FUNCTION_BLOCK AQ_SPLIT_2 (* Fan-Out: Splits 1 AQ into 2 AQ adapters *)
  (* Standard: 61499-2; Description: Copyright (c) 2026 Meisterschulen am Ostbahnhof SPDX-License-Identifier: EPL-2.0 *)
  (* Version 1.0, 2026-05-16, Franz Höpfinger, Meisterschulen am Ostbahnhof, Initial Version *)
  PACKAGE adapter::events::unidirectional;
  IMPORT eclipse4diac::core::GenericClassName;
  {SET_ATTRIBUTE(eclipse4diac::core::GenericClassName, 'GEN_AQ_SPLIT')}
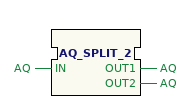
  SOCKETS
    IN : adapter::types::unidirectional::AQ; (* Input *)
  END_SOCKETS
  PLUGS
    OUT1 : adapter::types::unidirectional::AQ; (* Output 1 *)
    OUT2 : adapter::types::unidirectional::AQ; (* Output 2 *)
  END_PLUGS
END_FUNCTION_BLOCK
